PROGRAM MAIN
VAR
	counter1	:	FB_TestFunctionBlock;
END_VAR

counter1();

END_PROGRAM

(* stored: Version 1.1.0.1, ProductVersion 3.1.4024.11
   POU MAIN: Id {dbec18cf-ca82-4287-a487-95b423752fd7}, SpecialFunc None *)
